// TwinCAT 3 PLC project PRBS
// ProgramVersion: 3.1.4023.0
// libraries:
//   Tc2_Standard, * (Beckhoff Automation GmbH)
//   Tc2_System, * (Beckhoff Automation GmbH)
//   Tc3_Module, * (Beckhoff Automation GmbH)
// project tree:
//   DUTs/ E_System_Mode.TcDUT
//   / PlcTask.TcTTO
//   POUs/ FB_PRBS.TcPOU, MAIN.TcPOU
// real-time tasks:
//   TASK PlcTask: cycle T#10ms, priority 20, ADS port 350

CONFIGURATION PRBS
    RESOURCE PLC ON TwinCAT3
        TASK PlcTask(INTERVAL := T#10ms, PRIORITY := 20);
        PROGRAM MAIN WITH PlcTask : MAIN;
    END_RESOURCE
END_CONFIGURATION

// ---- DUTs/E_System_Mode.TcDUT
{attribute 'qualified_only'}
{attribute 'strict'}
TYPE E_System_Mode :
(
	System_Init := 0,
	System_Run
);
END_TYPE

// ---- POUs/MAIN.TcPOU
PROGRAM MAIN
VAR
END_VAR

END_PROGRAM

// ---- POUs/FB_PRBS.TcPOU
FUNCTION_BLOCK FB_PRBS
VAR_INPUT
	Mode	: 	E_System_Mode;	// current mode
	N 		: 	REAL;
	T 		: 	REAL;
	t_act	:	REAL;
	L 		: 	REAL;
	umin	: 	REAL;
	umax	: 	REAL;
END_VAR
VAR_OUTPUT
	u 		: 	REAL;
END_VAR
VAR
	reg 	: ARRAY [1..N] OF INT := 1; 
	k 		: LINT;
	sum 	: REAL;
END_VAR

CASE Mode OF
	E_System_Mode.System_Init:
	k := 1;
	sum := 0;
		
	E_System_Mode.System_Run:
	k := k + 1;
	
	CASE n OF
		2: 	sum := (reg[1]+reg[2]) MOD 2;
		3:	sum := (reg[2]+reg[3]) MOD 2;
		4:	sum := (reg[3]+reg[4]) MOD 2;
		5:	sum := (reg[5]+reg[3]) MOD 2;
		6:	sum := (reg[5]+reg[6]) MOD 2;
		7: 	sum := (reg[6]+reg[7]) MOD 2;
		8:	sum := (reg[4]+reg[5]+reg[6]+reg[8]) MOD 2;
		9:	sum := (reg[5]+reg[9]) MOD 2;
		10:	sum := (reg[7]+reg[10]) MOD 2;
		11:	sum := (reg[9]+reg[11]) MOD 2;
	END_CASE
	
	reg := SHR(reg, SIZEOF(reg));
	reg[1] = sum;
		
	ELSE  // default assignment
	;
		
END_CASE

END_FUNCTION_BLOCK
